# B&R Automation Studio project BaseLD
Automation Studio 4.7.2.98

## Configuration Config1

### Task classes (Cpu.sw)
```
Cyclic#4:
  Program <- Program.prg
  Program1 <- Program1.prg
```

### Hardware
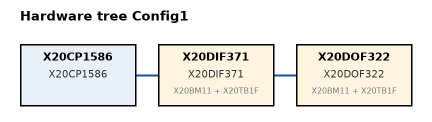
```
X20BM11a : X20BM11 v1.0.0.1  [X2X1 -> X20CP1586.IF6]
X20BM11b : X20BM11 v1.0.0.1  [X2X1 -> X20BM11a.X2X2]
X20CP1586 : X20CP1586 v1.8.0.0
X20DIF371 : X20DIF371 v1.1.0.0  [SS1 -> X20TB1F1.SS; SL -> X20BM11a.SL1]
X20DOF322 : X20DOF322 v1.3.0.0  [SS1 -> X20TB1F2.SS; SL -> X20BM11b.SL1]
X20TB1F1 : X20TB1F v1.0.0.0
X20TB1F2 : X20TB1F v1.0.0.0
```

## Logical view

### Program Logical/Program1 (IEC)

#### Variables.var
```iecst
VAR
	LEDon : BOOL;
	LEDoff : BOOL;
END_VAR
```

Listed in the project but not available here: Logical/Global.typ, Logical/Global.var, Logical/Libraries, Logical/Program
